KUKA KRL data list: Rack_Verde_CogerST121I.dat

&ACCESS RVO1
&REL 46
&COMMENT COGER ST121 RACK VERDE
&PARAM EDITMASK = *
&PARAM TEMPLATE = C:\KRC\Roboter\Template\vorgabe
&PARAM DISKPATH = KRC:\R1\Program\MAFELEC
DEFDAT  Rack_Verde_CogerST121I
;FOLD EXTERNAL DECLARATIONS;%{PE}%MKUKATPBASIS,%CEXT,%VCOMMON,%P
;FOLD GRIPPERTECH EXT
EXT  H50 (INT  :IN,INT  :IN,INT  :IN,GRP_TYP  :IN )
;ENDFOLD (GRIPPERTECH EXT)
;FOLD SPOTTECH EXT
EXT  USERSPOT (S_COMMAND  :IN,SPOT_TYPE  :IN )
;ENDFOLD (SPOTTECH EXT)
;FOLD BASISTECH EXT;%{PE}%MKUKATPBASIS,%CEXT,%VEXT,%P
EXT  BAS (BAS_COMMAND  :IN,REAL  :IN )
DECL INT SUCCESS
;ENDFOLD (BASISTECH EXT)
;FOLD USER EXT;%{E}%MKUKATPUSER,%CEXT,%VEXT,%P
;Make your modifications here

;ENDFOLD (USER EXT)
;ENDFOLD (EXTERNAL DECLARATIONS)
DECL BASIS_SUGG_T LAST_BASIS={POINT1[] "P0                      ",POINT2[] "P0                      ",CP_PARAMS[] "CPDAT0                  ",PTP_PARAMS[] "PDAT0                   ",CONT[] "                        ",CP_VEL[] "0.2                     ",PTP_VEL[] " 100                    ",SYNC_PARAMS[] "SYNCDAT                 ",SPL_NAME[] "S0                      ",A_PARAMS[] "ADAT0                   "}
DECL PDAT PH={VEL 100.000,ACC 100.000,APO_DIST 100.000,APO_MODE #CDIS,GEAR_JERK 50.0000,EXAX_IGN 0}
DECL E6POS XP10={X 475.302704,Y 670.277710,Z 581.127319,A 179.609329,B -0.271935076,C 179.783524,S 2,T 10,E1 0.0,E2 0.0,E3 0.0,E4 0.0,E5 0.0,E6 0.0}
DECL FDAT FP10={TOOL_NO 9,BASE_NO 3,IPO_FRAME #BASE,POINT2[] " ",TQ_STATE FALSE}
DECL E6POS XP20={X 475.302704,Y 670.277710,Z 75.6043396,A 179.609329,B -0.271935076,C 179.783524,S 2,T 10,E1 0.0,E2 0.0,E3 0.0,E4 0.0,E5 0.0,E6 0.0}
DECL FDAT FP20={TOOL_NO 9,BASE_NO 3,IPO_FRAME #BASE,POINT2[] " ",TQ_STATE FALSE}
DECL E6POS XPOS_COGER_ST121={X 585.103516,Y 632.197,Z 39.5193100,A 179.699509,B -0.370581716,C 179.870728,S 2,T 10,E1 0.0,E2 0.0,E3 0.0,E4 0.0,E5 0.0,E6 0.0}
DECL FDAT FPos_Coger_ST121={TOOL_NO 9,BASE_NO 3,IPO_FRAME #BASE,POINT2[] " ",TQ_STATE FALSE}
DECL PDAT PM={VEL 100.000,ACC 50.0000,APO_DIST 50.0000,APO_MODE #CDIS,GEAR_JERK 50.0000,EXAX_IGN 0}
DECL E6POS XPOS_ESPERA_ST121={X 1597.05444,Y -395.116150,Z 1941.31274,A -176.307449,B 30.3077869,C -171.065643,S 2,T 10,E1 0.0,E2 0.0,E3 0.0,E4 0.0,E5 0.0,E6 0.0}
DECL FDAT FPOS_ESPERA_ST121={TOOL_NO 9,BASE_NO 0,IPO_FRAME #BASE,POINT2[] " ",TQ_STATE FALSE}
DECL LDAT LM={VEL 2.00000,ACC 25.0000,APO_DIST 100.000,APO_FAC 50.0000,AXIS_VEL 100.000,AXIS_ACC 100.000,ORI_TYP #VAR,CIRC_TYP #BASE,JERK_FAC 50.0000,GEAR_JERK 50.0000,EXAX_IGN 0}
DECL E6POS XPOS_SOBRE_ST121={X 475.302704,Y 670.277710,Z 348.834778,A 179.609329,B -0.271935076,C 179.783524,S 2,T 10,E1 0.0,E2 0.0,E3 0.0,E4 0.0,E5 0.0,E6 0.0}
DECL FDAT FPOS_SOBRE_ST121={TOOL_NO 11,BASE_NO 3,IPO_FRAME #BASE,POINT2[] " ",TQ_STATE FALSE}
DECL E6POS XPOS_SOBRE_ST122={X 1790.32410,Y 1.34322268E-13,Z 1909.62585,A -180.000,B 89.9853210,C -180.000,S 2,T 3,E1 0.0,E2 0.0,E3 0.0,E4 0.0,E5 0.0,E6 0.0}
DECL FDAT FPOS_SOBRE_ST122={TOOL_NO 9,BASE_NO 3,IPO_FRAME #BASE,POINT2[] " ",TQ_STATE FALSE}
DECL E6POS XP30={X -507.111389,Y 1063.31885,Z 760.188049,A -47.6190376,B -0.167292342,C 179.537186,S 2,T 34,E1 0.0,E2 0.0,E3 0.0,E4 0.0,E5 0.0,E6 0.0}
DECL FDAT FP30={TOOL_NO 11,BASE_NO 3,IPO_FRAME #BASE,POINT2[] " ",TQ_STATE FALSE}
DECL E6POS XP40={X -0.0319372341,Y -2.62910700,Z -362.053223,A -0.00123304490,B -0.0257057231,C 0.00384289422,S 2,T 10,E1 0.0,E2 0.0,E3 0.0,E4 0.0,E5 0.0,E6 0.0}
DECL FDAT FP40={TOOL_NO 11,BASE_NO 3,IPO_FRAME #BASE,POINT2[] " ",TQ_STATE FALSE}
DECL E6POS XPOS_AREA_3_LIBRE={X 772.101379,Y -764.727417,Z 1373.18774,A -87.1007538,B -0.167297110,C 179.537186,S 2,T 34,E1 0.0,E2 0.0,E3 0.0,E4 0.0,E5 0.0,E6 0.0}
DECL FDAT FPOS_AREA_3_LIBRE={TOOL_NO 11,BASE_NO 0,IPO_FRAME #BASE,POINT2[] " ",TQ_STATE FALSE}
DECL GRP_SUGG_T LAST_GRP={NUMBER[] "1                       ",STATE[] "1                       ",PARAMS[] "GDAT0                   "}
DECL LDAT LL={VEL 2.00000,ACC 25.0000,APO_DIST 100.000,APO_FAC 50.0000,AXIS_VEL 100.000,AXIS_ACC 100.000,ORI_TYP #VAR,CIRC_TYP #BASE,JERK_FAC 50.0000,GEAR_JERK 50.0000,EXAX_IGN 0}
DECL E6POS XPOS_COGER_AZUL_ST121={X 431.750763,Y 643.881836,Z 37.8616257,A -0.404950738,B 0.00806899648,C -179.935089,S 2,T 42,E1 0.0,E2 0.0,E3 0.0,E4 0.0,E5 0.0,E6 0.0}
DECL FDAT FPos_Coger_Azul_ST121={TOOL_NO 9,BASE_NO 3,IPO_FRAME #BASE,POINT2[] " ",TQ_STATE FALSE}
DECL E6POS XPOS_WAIT_VERDE_ST121={X 1606.70789,Y -354.796814,Z 1944.22656,A 1.33749425,B -32.3921471,C 179.037674,S 2,T 42,E1 0.0,E2 0.0,E3 0.0,E4 0.0,E5 0.0,E6 0.0}
DECL FDAT FPOS_Wait_Verde_ST121={TOOL_NO 9,BASE_NO 0,IPO_FRAME #BASE,POINT2[] " ",TQ_STATE FALSE}
DECL E6POS XPos_Coger_Verde_ST121={X 364.233917,Y 680.820,Z 35.4071388,A -0.219467372,B -0.287552029,C -179.748962,S 2,T 42,E1 0.0,E2 0.0,E3 0.0,E4 0.0,E5 0.0,E6 0.0}
DECL FDAT FPos_Coger_Verde_ST121={TOOL_NO 9,BASE_NO 3,IPO_FRAME #BASE,POINT2[] " ",TQ_STATE FALSE}
DECL PDAT PL={VEL 100.000,ACC 50.0000,APO_DIST 50.0000,APO_MODE #CDIS,GEAR_JERK 50.0000,EXAX_IGN 0}
DECL E6POS XP0={X 312.450226,Y 675.070,Z 407.579834,A -0.219463497,B -0.287549138,C -179.748962,S 2,T 42,E1 0.0,E2 0.0,E3 0.0,E4 0.0,E5 0.0,E6 0.0}
DECL FDAT FP0={TOOL_NO 9,BASE_NO 3,IPO_FRAME #BASE,POINT2[] " ",TQ_STATE FALSE}
DECL E6POS XP1={X 312.450226,Y 675.070,Z 73.4258270,A -0.219463497,B -0.287549138,C -179.748962,S 2,T 42,E1 0.0,E2 0.0,E3 0.0,E4 0.0,E5 0.0,E6 0.0}
DECL FDAT FP1={TOOL_NO 9,BASE_NO 3,IPO_FRAME #BASE,POINT2[] " ",TQ_STATE FALSE}
DECL E6POS XCoger_ST121_INSP={X 312.450226,Y 675.070,Z 35.5267525,A -0.219463542,B -0.287549138,C -179.748962,S 2,T 42,E1 0.0,E2 0.0,E3 0.0,E4 0.0,E5 0.0,E6 0.0}
DECL FDAT FCoger_ST121_INSP={TOOL_NO 9,BASE_NO 3,IPO_FRAME #BASE,POINT2[] " ",TQ_STATE FALSE}
DECL E6POS XCoger_Verde_ST121_INSP={X 475.302704,Y 670.277710,Z 29.8382587,A 179.609329,B -0.271935105,C 179.783524,S 2,T 10,E1 0.0,E2 0.0,E3 0.0,E4 0.0,E5 0.0,E6 0.0}
DECL FDAT FCoger_Verde_ST121_INSP={TOOL_NO 9,BASE_NO 3,IPO_FRAME #BASE,POINT2[] " ",TQ_STATE FALSE}
DECL E6POS XPOS_SOBRE_ST123={X 475.302704,Y 670.277710,Z 348.834778,A 179.609329,B -0.271935076,C 179.783524,S 2,T 10,E1 0.0,E2 0.0,E3 0.0,E4 0.0,E5 0.0,E6 0.0}
DECL FDAT FPOS_SOBRE_ST123={TOOL_NO 11,BASE_NO 3,IPO_FRAME #BASE,POINT2[] " ",TQ_STATE FALSE}
ENDDAT
